{attribute 'GeneratedUsingTerminal: EL9195--0000'}
{attribute addProperty BoxType "EL9195--0000"}
{attribute addProperty Description "EL9195 Potential Connection, 2 x Shield"}
{attribute addProperty Physics "KK"}
{attribute addProperty Id "EL9195"}
{attribute addProperty CRC "1321837627"}
{attribute addProperty Size "0"}
TYPE EL9195_4EC9A43B EXTENDS EtcSlaveTerminalBase_947E5A46 :
STRUCT
END_STRUCT
END_TYPE

(* stored: Version 1.2.0.0, ProductVersion 3.1.4024.11
   DUT EL9195_4EC9A43B: Id {357aa243-8724-495c-a913-873a9dc417b9} *)
